// TIA Portal V17 export
// export: Created 2022-03-12T16:05:29.806558Z, ExportSetting WithDefaults, DisplayName Totally Integrated Automation Portal, DisplayVersion V17, DisplayName TIA Portal Openness, DisplayVersion V17, DisplayName TIA Portal Version Control Interface, DisplayVersion V17, DisplayName STEP 7 Professional, DisplayVersion V17, DisplayName STEP 7 Safety, DisplayVersion V17, DisplayName WinCC Advanced / Unified PC, DisplayVersion V17
DATA_BLOCK "PackMLCfg"   // DB31603
TITLE = CPG_PackMLCfg
{ S7_Optimized_Access := 'TRUE' }
AUTHOR : tech.team.motioncontrol@siemens.com
FAMILY : CPG
VERSION : 1.0
// Support: tech.team.motioncontrol@siemens.com
// Fax: +49 (0) 9131/98-1297
// stored: AutoNumber true, DBAccessibleFromOPCUA true, DBAccessibleFromWebserver true, IsOnlyStoredInLoadMemory false, IsRetainMemResEnabled false, IsWriteProtectedInAS false, MemoryReserve 0
   VAR
      Cfg { S7_SetPoint := 'True'} : "typeLPMLV30_Configuration";   // PackML Configuration Data
      Names { S7_SetPoint := 'True'} : "typeLPMLV30_NamesConfiguration";   // PackML Names Data
      disable : Struct   // Bits used to disable TR88 UN & EMs
         UN : Bool;   // UN (1 = disable, 0= enable)
         EM00 : Struct   // EM00 (1 = disable, 0 = enable)
            EM : Bool;   // EMxx (1 = disable, 0 = enable)
            CM01 : Bool;   // CMxx (1 = disable, 0 = enable)
            CM02 : Bool;   // CMxx (1 = disable, 0 = enable)
            CM03 : Bool;   // CMxx (1 = disable, 0 = enable)
            CM04 : Bool;   // CMxx (1 = disable, 0 = enable)
            CM05 : Bool;   // CMxx (1 = disable, 0 = enable)
            CM06 : Bool;   // CMxx (1 = disable, 0 = enable)
            CM07 : Bool;   // CMxx (1 = disable, 0 = enable)
            CM08 : Bool;   // CMxx (1 = disable, 0 = enable)
            CM09 : Bool;   // CMxx (1 = disable, 0 = enable)
            CM10 : Bool;   // CMxx (1 = disable, 0 = enable)
         END_STRUCT;
         EM01 : Struct   // EM01 (1 = disable, 0 = enable)
            EM : Bool;   // EMxx (1 = disable, 0 = enable)
            CM01 : Bool;   // CMxx (1 = disable, 0 = enable)
            CM02 : Bool;   // CMxx (1 = disable, 0 = enable)
            CM03 : Bool;   // CMxx (1 = disable, 0 = enable)
            CM04 : Bool;   // CMxx (1 = disable, 0 = enable)
            CM05 : Bool;   // CMxx (1 = disable, 0 = enable)
            CM06 : Bool;   // CMxx (1 = disable, 0 = enable)
            CM07 : Bool;   // CMxx (1 = disable, 0 = enable)
            CM08 : Bool;   // CMxx (1 = disable, 0 = enable)
            CM09 : Bool;   // CMxx (1 = disable, 0 = enable)
            CM10 : Bool;   // CMxx (1 = disable, 0 = enable)
         END_STRUCT;
         EM02 : Struct   // EM02 (1 = disable, 0 = enable)
            EM : Bool;   // EMxx (1 = disable, 0 = enable)
            CM01 : Bool;   // CMxx (1 = disable, 0 = enable)
            CM02 : Bool;   // CMxx (1 = disable, 0 = enable)
            CM03 : Bool;   // CMxx (1 = disable, 0 = enable)
            CM04 : Bool;   // CMxx (1 = disable, 0 = enable)
            CM05 : Bool;   // CMxx (1 = disable, 0 = enable)
            CM06 : Bool;   // CMxx (1 = disable, 0 = enable)
            CM07 : Bool;   // CMxx (1 = disable, 0 = enable)
            CM08 : Bool;   // CMxx (1 = disable, 0 = enable)
            CM09 : Bool;   // CMxx (1 = disable, 0 = enable)
            CM10 : Bool;   // CMxx (1 = disable, 0 = enable)
         END_STRUCT;
         EM03 : Struct   // EM03 (1 = disable, 0 = enable)
            EM : Bool;   // EMxx (1 = disable, 0 = enable)
            CM01 : Bool;   // CMxx (1 = disable, 0 = enable)
            CM02 : Bool;   // CMxx (1 = disable, 0 = enable)
            CM03 : Bool;   // CMxx (1 = disable, 0 = enable)
            CM04 : Bool;   // CMxx (1 = disable, 0 = enable)
            CM05 : Bool;   // CMxx (1 = disable, 0 = enable)
            CM06 : Bool;   // CMxx (1 = disable, 0 = enable)
            CM07 : Bool;   // CMxx (1 = disable, 0 = enable)
            CM08 : Bool;   // CMxx (1 = disable, 0 = enable)
            CM09 : Bool;   // CMxx (1 = disable, 0 = enable)
            CM10 : Bool;   // CMxx (1 = disable, 0 = enable)
         END_STRUCT;
         EM04 : Struct   // EM04 (1 = disable, 0 = enable)
            EM : Bool;   // EMxx (1 = disable, 0 = enable)
            CM01 : Bool;   // CMxx (1 = disable, 0 = enable)
            CM02 : Bool;   // CMxx (1 = disable, 0 = enable)
            CM03 : Bool;   // CMxx (1 = disable, 0 = enable)
            CM04 : Bool;   // CMxx (1 = disable, 0 = enable)
            CM05 : Bool;   // CMxx (1 = disable, 0 = enable)
            CM06 : Bool;   // CMxx (1 = disable, 0 = enable)
            CM07 : Bool;   // CMxx (1 = disable, 0 = enable)
            CM08 : Bool;   // CMxx (1 = disable, 0 = enable)
            CM09 : Bool;   // CMxx (1 = disable, 0 = enable)
            CM10 : Bool;   // CMxx (1 = disable, 0 = enable)
         END_STRUCT;
         EM05 : Struct   // EM05 (1 = disable, 0 = enable)
            EM : Bool;   // EMxx (1 = disable, 0 = enable)
            CM01 : Bool;   // CMxx (1 = disable, 0 = enable)
            CM02 : Bool;   // CMxx (1 = disable, 0 = enable)
            CM03 : Bool;   // CMxx (1 = disable, 0 = enable)
            CM04 : Bool;   // CMxx (1 = disable, 0 = enable)
            CM05 : Bool;   // CMxx (1 = disable, 0 = enable)
            CM06 : Bool;   // CMxx (1 = disable, 0 = enable)
            CM07 : Bool;   // CMxx (1 = disable, 0 = enable)
            CM08 : Bool;   // CMxx (1 = disable, 0 = enable)
            CM09 : Bool;   // CMxx (1 = disable, 0 = enable)
            CM10 : Bool;   // CMxx (1 = disable, 0 = enable)
         END_STRUCT;
         EM06 : Struct   // EM06 (1 = disable, 0 = enable)
            EM : Bool;   // EMxx (1 = disable, 0 = enable)
            CM01 : Bool;   // CMxx (1 = disable, 0 = enable)
            CM02 : Bool;   // CMxx (1 = disable, 0 = enable)
            CM03 : Bool;   // CMxx (1 = disable, 0 = enable)
            CM04 : Bool;   // CMxx (1 = disable, 0 = enable)
            CM05 : Bool;   // CMxx (1 = disable, 0 = enable)
            CM06 : Bool;   // CMxx (1 = disable, 0 = enable)
            CM07 : Bool;   // CMxx (1 = disable, 0 = enable)
            CM08 : Bool;   // CMxx (1 = disable, 0 = enable)
            CM09 : Bool;   // CMxx (1 = disable, 0 = enable)
            CM10 : Bool;   // CMxx (1 = disable, 0 = enable)
         END_STRUCT;
         EM07 : Struct   // EM07 (1 = disable, 0 = enable)
            EM : Bool;   // EMxx (1 = disable, 0 = enable)
            CM01 : Bool;   // CMxx (1 = disable, 0 = enable)
            CM02 : Bool;   // CMxx (1 = disable, 0 = enable)
            CM03 : Bool;   // CMxx (1 = disable, 0 = enable)
            CM04 : Bool;   // CMxx (1 = disable, 0 = enable)
            CM05 : Bool;   // CMxx (1 = disable, 0 = enable)
            CM06 : Bool;   // CMxx (1 = disable, 0 = enable)
            CM07 : Bool;   // CMxx (1 = disable, 0 = enable)
            CM08 : Bool;   // CMxx (1 = disable, 0 = enable)
            CM09 : Bool;   // CMxx (1 = disable, 0 = enable)
            CM10 : Bool;   // CMxx (1 = disable, 0 = enable)
         END_STRUCT;
         EM08 : Struct   // EM08 (1 = disable, 0 = enable)
            EM : Bool;   // EMxx (1 = disable, 0 = enable)
            CM01 : Bool;   // CMxx (1 = disable, 0 = enable)
            CM02 : Bool;   // CMxx (1 = disable, 0 = enable)
            CM03 : Bool;   // CMxx (1 = disable, 0 = enable)
            CM04 : Bool;   // CMxx (1 = disable, 0 = enable)
            CM05 : Bool;   // CMxx (1 = disable, 0 = enable)
            CM06 : Bool;   // CMxx (1 = disable, 0 = enable)
            CM07 : Bool;   // CMxx (1 = disable, 0 = enable)
            CM08 : Bool;   // CMxx (1 = disable, 0 = enable)
            CM09 : Bool;   // CMxx (1 = disable, 0 = enable)
            CM10 : Bool;   // CMxx (1 = disable, 0 = enable)
         END_STRUCT;
         EM09 : Struct   // EM09 (1 = disable, 0 = enable)
            EM : Bool;   // EMxx (1 = disable, 0 = enable)
            CM01 : Bool;   // CMxx (1 = disable, 0 = enable)
            CM02 : Bool;   // CMxx (1 = disable, 0 = enable)
            CM03 : Bool;   // CMxx (1 = disable, 0 = enable)
            CM04 : Bool;   // CMxx (1 = disable, 0 = enable)
            CM05 : Bool;   // CMxx (1 = disable, 0 = enable)
            CM06 : Bool;   // CMxx (1 = disable, 0 = enable)
            CM07 : Bool;   // CMxx (1 = disable, 0 = enable)
            CM08 : Bool;   // CMxx (1 = disable, 0 = enable)
            CM09 : Bool;   // CMxx (1 = disable, 0 = enable)
            CM10 : Bool;   // CMxx (1 = disable, 0 = enable)
         END_STRUCT;
      END_STRUCT;
   END_VAR
BEGIN
   Names.unitModesNames[2,0] := 'Invalid';
   Names.unitModesNames[2,1] := 'Production';
   Names.unitModesNames[2,2] := 'Maintenance';
   Names.unitModesNames[2,3] := 'Manual';
   Names.unitModesNames[2,4] := 'User Mode 01';
   Names.statesNames[1,1] := 'Clearing';
   Names.statesNames[1,2] := 'Stopped';
   Names.statesNames[1,3] := 'Starting';
   Names.statesNames[1,4] := 'Idle';
   Names.statesNames[1,5] := 'Suspended';
   Names.statesNames[1,6] := 'Execute';
   Names.statesNames[1,7] := 'Stopping';
   Names.statesNames[1,8] := 'Aborting';
   Names.statesNames[1,9] := 'Aborted';
   Names.statesNames[1,10] := 'Holding';
   Names.statesNames[1,11] := 'Held';
   Names.statesNames[1,12] := 'UnHolding';
   Names.statesNames[1,13] := 'Suspending';
   Names.statesNames[1,14] := 'UnSuspending';
   Names.statesNames[1,15] := 'Resetting';
   Names.statesNames[1,16] := 'Completing';
   Names.statesNames[1,17] := 'Complete';
   Names.statesNames[2,0] := 'Undefined';
   Names.statesNames[2,1] := 'Limpiar';
   Names.statesNames[2,2] := 'Detenido';
   Names.statesNames[2,3] := 'Empezando';
   Names.statesNames[2,4] := 'Parado';
   Names.statesNames[2,5] := 'Interrumpido';
   Names.statesNames[2,6] := 'Correr';
   Names.statesNames[2,7] := 'Detener';
   Names.statesNames[2,8] := 'Anulando';
   Names.statesNames[2,9] := 'Anulado';
   Names.statesNames[2,10] := 'Mantener';
   Names.statesNames[2,11] := 'Mantenido';
   Names.statesNames[2,12] := 'Desmentener';
   Names.statesNames[2,13] := 'Interrumpir';
   Names.statesNames[2,14] := 'Desinterrumpir';
   Names.statesNames[2,15] := 'Reajustar';
   Names.statesNames[2,16] := 'Terminar';
   Names.statesNames[2,17] := 'Terminado';
END_DATA_BLOCK
